TYPE ST_SequenceItem :
STRUCT
	nId			: UINT;
	nValue		: USINT(0..100);
	nDuration	: UINT;
END_STRUCT
END_TYPE

(* stored: Version 1.1.0.1, ProductVersion 3.1.4024.12
   DUT ST_SequenceItem: Id {bca356fa-a85b-42fc-ae20-b35eb146e406} *)
